// TIA Portal V19 export
FUNCTION "DTrk_DeleteAll" : Void   // FC166, LAD
// stored: SetENOAutomatically false
BEGIN

REGION Network 1
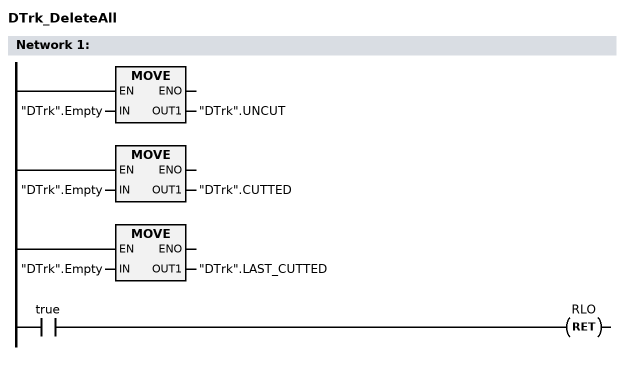
   "DTrk".UNCUT := "DTrk".Empty;
   "DTrk".CUTTED := "DTrk".Empty;
   "DTrk".LAST_CUTTED := "DTrk".Empty;
   IF true THEN
       ENO := TRUE;
       RETURN;
   END_IF;
END_REGION
END_FUNCTION
